{attribute 'qualified_only'}
VAR_GLOBAL
	fJoystickNormalizedY 		: LREAL; 
	fJoystickNormalizedX 		: LREAL; 
	fJoystickNormalizedZ 		: LREAL; 
	fPressureWinchA1 	 		: LREAL; 
	fPressureWinchA2 	 		: LREAL; 
	fPressureWinchB 	 		: LREAL; 
	fPressureCylinderA 	 		: LREAL;  
	fPressureCylinderB 	 		: LREAL; 
	fPressureSupply 	 		: LREAL; 
	fPressureReturn 	 		: LREAL; 
	fWinchEncoderPosition 		: LREAL;
	fCylinderEncoderPosition 	: LREAL;
	fCylinderPosition 			:LREAL;
END_VAR

(* stored: Version 1.1.0.1, ProductVersion 3.1.4024.12
   GVL G_Sensors: Id {4ff3b0b3-7afb-45b2-8b55-d797c734f296} *)
